(* Logix 5000 project; controller KTC_tresure vendor 1 type 14 code 149 rev 30.11; software revision 30.00 *)

TASK MainTask (continuous, watchdog 500 ms) : MainProgram

MODULES
   Local : vendor 1 type 14 code 149 (Compact 0, rev 30.11)
      Discrete_IO : Embedded (Compact 1, rev 3.1, Output RPI 20 ms)
END_MODULES

PROGRAM MainProgram   (* main routine MainRoutine *)
VAR
   blues : BOOL;
   pb1 : ALIAS FOR Local:1:I.Data.0;   // tresure on red
   pb2 : ALIAS FOR Local:1:I.Data.1;   // tresure on blue
   pb3 : ALIAS FOR Local:1:I.Data.5;   // end position blue
   pb4 : ALIAS FOR Local:1:I.Data.3;   // start position blue
   pb5 : ALIAS FOR Local:1:I.Data.4;   // start positon red
   pb6 : ALIAS FOR Local:1:I.Data.6;   // end position red
   pb7 : ALIAS FOR Local:1:I.Data.2;   // both bars
   sol1 : ALIAS FOR Local:1:O.Data.0;   // move red
   sol2 : ALIAS FOR Local:1:O.Data.1;   // move blue
   sol3 : ALIAS FOR Local:1:O.Data.4;   // mark
   sol4 : ALIAS FOR Local:1:O.Data.3;   // switch direction blue
   sol5 : ALIAS FOR Local:1:O.Data.2;   // switch direction red
END_VAR

ROUTINE MainRoutine   (* ladder *)
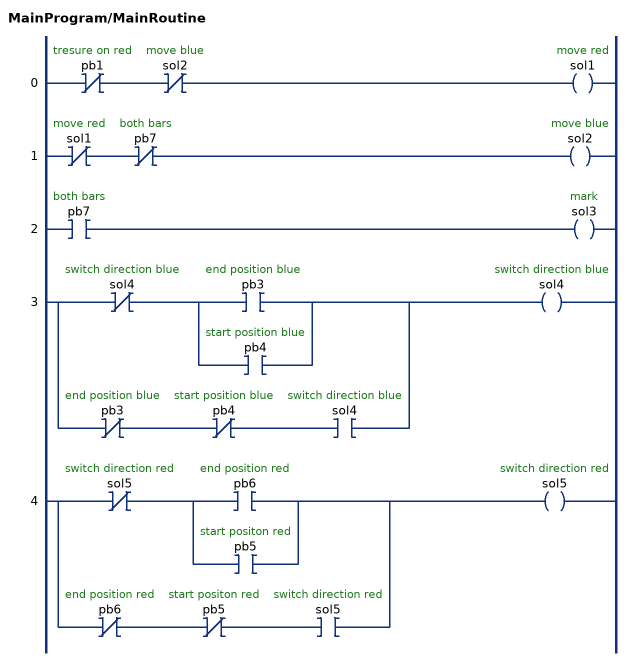
   0: XIO(pb1)XIO(sol2)OTE(sol1);
   1: XIO(sol1)XIO(pb7)OTE(sol2);
   2: XIC(pb7)OTE(sol3);
   3: [XIO(sol4) [XIC(pb3) ,XIC(pb4) ] ,XIO(pb3) XIO(pb4) XIC(sol4) ]OTE(sol4);
   4: [XIO(sol5) [XIC(pb6) ,XIC(pb5) ] ,XIO(pb6) XIO(pb5) XIC(sol5) ]OTE(sol5);
END_ROUTINE
END_PROGRAM
